INTERFACE IEventHandler_OnHourChanged EXTENDS IEventHandlerBase

METHOD OnHourChanged
VAR_INPUT
	Now: TIMESTRUCT;
END_VAR
END_METHOD

END_INTERFACE

(* stored: Version 1.1.0.1, ProductVersion 3.1.4024.3
   Itf IEventHandler_OnHourChanged: Id {f2f56ecb-2c7b-0ae7-3fe5-f8bb552022a0}
   Method OnHourChanged: Id {ca9b7a78-0305-0243-19c3-14e62fe67cfb} *)
